FUNCTION_BLOCK ABSTRACT FileHandleTask EXTENDS TOF_Tasks.Task IMPLEMENTS IFileHandleTask
VAR
	_FileOpen : REFERENCE TO Tc2_System.FB_FileOpen;
END_VAR

{attribute 'monitoring' := 'call'}
PROPERTY ABSTRACT AmsNetId : Tc2_System.T_AmsNetID
GET
END_GET
SET
END_SET
END_PROPERTY

{attribute 'monitoring' := 'call'}
PROPERTY FINAL FileHandle : UINT
GET
IF __ISVALIDREF(_FileOpen) THEN
	FileHandle := _FileOpen.hFile;
END_IF
END_GET
END_PROPERTY

{attribute 'monitoring' := 'call'}
PROPERTY FINAL FilePath : Tc2_System.T_MaxString
GET
IF __ISVALIDREF(_FileOpen) THEN
	FilePath := _FileOpen.sPathName;
END_IF
END_GET
END_PROPERTY

METHOD SetFileOpen
VAR_INPUT
	fileOpen : REFERENCE TO Tc2_System.FB_FileOpen;
END_VAR
_FileOpen REF= fileOpen;
END_METHOD

{attribute 'monitoring' := 'call'}
{attribute 'OPC.UA.DA.Property' := '1'}
{attribute 'OPC.UA.DA' := '1'}
PROPERTY ABSTRACT Timeout : TIME
GET
END_GET
SET
END_SET
END_PROPERTY

END_FUNCTION_BLOCK

(* stored: Version 1.1.0.1
   POU FileHandleTask: Id {e0edebf6-69ee-43f1-b0cd-ddf0e5a3f8d2}, SpecialFunc None
   Property AmsNetId: Id {ea169d19-fc59-4e8e-bfd6-f05e2562e2f5}
   Get Get: Id {75d6b396-2e53-497e-98ab-b2564567cddb}
   Set Set: Id {94e4e0c9-5dda-4170-b1e7-d631abb75196}
   Property FileHandle: Id {82868fbc-d80b-4342-95ff-b87334c6f19e}
   Get Get: Id {00add956-e3ac-47c9-87bd-7a30ec1b127b}
   Property FilePath: Id {5eefa187-b2a6-4167-b37b-7a1237013146}
   Get Get: Id {b73f03f2-fbb8-4ef6-a600-eed689f598d3}
   Method SetFileOpen: Id {ae64e717-44da-42dc-b4c5-bc1e2b25543b}
   Property Timeout: Id {b3334de9-562b-4b05-996c-bb7c42bd5ba7}
   Get Get: Id {35a70dd8-7700-4e7d-a505-0a238f1252c8}
   Set Set: Id {833a7c4a-0925-4e43-965f-120e0cbe7c74} *)
